// TwinCAT 3 PLC project reading_plc_proj
// ProgramVersion: 3.1.4023.0
// libraries:
//   L2SI Vacuum Library, * (SLAC)
//   LCLS General, * (SLAC)
//   Tc2_Standard, * (Beckhoff Automation GmbH)
//   Tc2_System, * (Beckhoff Automation GmbH)
//   Tc3_Module, * (Beckhoff Automation GmbH)
// project tree:
//   / PlcTask.TcTTO
//   POUs/ MAIN.TcPOU
// real-time tasks:
//   TASK PlcTask: cycle T#10ms, priority 20, ADS port 350

CONFIGURATION reading_plc_proj
    RESOURCE PLC ON TwinCAT3
        TASK PlcTask(INTERVAL := T#10ms, PRIORITY := 20);
        PROGRAM MAIN WITH PlcTask : MAIN;
    END_RESOURCE
END_CONFIGURATION

// ---- POUs/MAIN.TcPOU
PROGRAM MAIN
VAR
	counter_x : INT;
	
	vgc_reader : FB_TVGC_ADS;
	gcc_reader : FB_TGCC_ADS;
	
END_VAR

// A counter to confirm that the program is running
counter_x := counter_x + 1;

END_PROGRAM
